//--
// <ObjectWithoutContextExampleDeclaration>
(*
		
			This is an example of self-confident object, that initiate its context by itself.

*)
FUNCTION_BLOCK Woltz_Object EXTENDS Person_Object
VAR
	//Horse owned by Jack Woltz.
	//https://godfather.fandom.com/wiki/Khartoum
	_Khartoum	: Horse_Object(THIS^);
END_VAR
//---------------------------------------------------------------------------
// </ObjectWithoutContextExampleDeclaration>
//--

END_FUNCTION_BLOCK

(* stored: Version 1.1.0.1, ProductVersion 3.1.4024.6
   POU Woltz_Object: Id {210d7878-f3a8-0d74-1c18-c55600d21082}, SpecialFunc None *)
